FUNCTION_BLOCK SubMachine2 extends Composite
VAR
	component1					: Component;
	component2					: Component;
	component3					: Component;
	childs						: ARRAY[1..NOOFCHILDS] OF IComposite := [component1,component2,component3]; 	
END_VAR
VAR CONSTANT
	NOOFCHILDS					: INT := 3;
END_VAR

METHOD logStatus
VAR
	sMessage				: STRING;		
	i						: DINT;
END_VAR
// Local status 
SUPER^.logStatus();

// Loop through childs
FOR i := 1 TO NOOFCHILDS DO
	IF childs[i]<>0 THEN
		childs[i].logStatus();
	END_IF
END_FOR
END_METHOD

END_FUNCTION_BLOCK

(* stored: Version 1.1.0.1, ProductVersion 3.1.4024.12
   POU SubMachine2: Id {3dc6a06c-5ad5-4410-a5bf-aef531f5e96a}, SpecialFunc None
   Method logStatus: Id {db797f28-bedb-45ec-b58e-88eb34e00ed2} *)
